// TIA Portal V20 export
VAR_GLOBAL   // PLC tag table "Standard-Variablentabelle"
END_VAR
